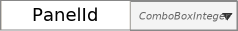
VISUALIZATION V_AkPanelSelecCmb  // 238x31
    ComboBoxInteger (130,1 108x30), variable: VisuGVL.fbPanelImp.AKPanelId, text list: 'AkCmbTxtList'
    Textfield (1,0 129x30), "PanelId"
END_VISUALIZATION

(* stored: Version 1.1.0.1, ProductVersion 3.1.4024.4
   Visu V_AkPanelSelecCmb: Id {0e5a8c85-5538-4d64-8650-3eaed8def088} *)
